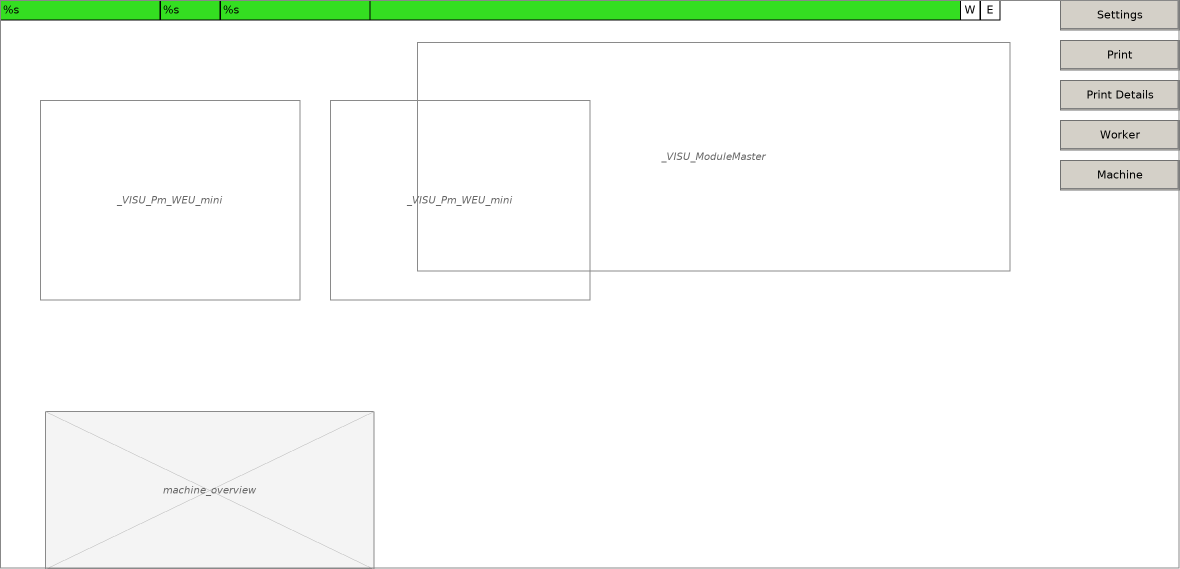
VISUALIZATION VISU_PrintOverview  // 1180x569, background image calmar_bg
    Image (45,411 329x158), image: machine_overview
    Rectangle (0,0 1000x20)
    Button (1060,0 120x30), "Settings"
        OnMouseClick: change screen: VISU_SettingsWeu
    Button (1060,40 120x30), "Print"
        OnMouseClick: change screen: VISU_PRINT
    Button (1060,80 120x30), "Print Details"
        OnMouseClick: change screen: VISU_PrintDetails
    Button (1060,120 120x30), "Worker"
        OnMouseClick: change screen: VISU_Workers
    Frame (417,42 593x229)
        shows _VISU_ModuleMaster(mInst := PRG_PRINT.fbModuleMaster)
    Rectangle (220,0 150x20), "%s", tooltip "Date & Time", text variable: PRG_SYSTEM.aCurrentDateTime
    Rectangle (0,0 160x20), "%s", tooltip "Project", text variable: PRG_SYSTEM.sC_Ads_System.aProject
    RoundedRectangle (980,0 20x20), "E", tooltip "Error Message active"
        toggle PRG_MACHINE.bO_ErrorMsgActive
    RoundedRectangle (960,0 20x20), "W", tooltip "Warning Message active"
        toggle PRG_MACHINE.bO_WarningMsgActive
    Rectangle (160,0 60x20), "%s", tooltip "Project", text variable: PRG_SYSTEM.sC_Ads_System.aMachine
    Frame (330,100 260x200)
        shows _VISU_Pm_WEU_mini(mInst := PRG_PRINT.fbPrintModule[1])
    Frame (40,100 260x200)
        shows _VISU_Pm_WEU_mini(mInst := PRG_PRINT.fbPrintModule[2])
    Button (1060,160 120x30), "Machine"
        OnMouseClick: change screen: VISU_MACHINE
END_VISUALIZATION

(* stored: Version 1.1.0.1, ProductVersion 3.1.4024.11
   Visu VISU_PrintOverview: Id {a6ed15b6-9f2e-485d-8015-919bd40398e8} *)
